// TIA Portal V20 export
TYPE "typeMainOpMode"
// stored: Access Published, IsFailsafeCompliant true, Namespace Safety
   STRUCT
      auto : Bool;   // Auto Mode
      manual : Bool;   // Manual Mode
      home : Bool;   // Auto Ready Start
      reset : Bool;   // Safety Reset
      enable : Bool;   // OP_Enable
   END_STRUCT;
END_TYPE
